TYPE "MES_Err_&_Msg"
VERSION : 0.1
// Block: MES_Err_&_Msg
   STRUCT
      Presence : Bool;
      Code : DInt;
      Description : String;
      Msg : MES_Msg;
   END_STRUCT;

END_TYPE
